Yaskawa INFORM job: TEST_KR.JBI

/JOB
//NAME TEST_KR
///FOLDERNAME INNE
//POS
///NPOS 2,2,0,0,0,0
///TOOL 0
///POSTYPE ROBOT
///RECTAN
///RCONF 0,0,0,0,0,0,0,0,0,0,0,0,0,0,0,0,0,0,0,0,0,0,0,0
C00000=-1082.109,-1268.604,-1687.249,-50.7166,43.0014,-29.7739
C00001=-1082.109,-1268.604,-1687.249,-50.7166,43.0014,-29.7739
BC00000=2160.163,372.281,1842.609
BC00001=2160.163,372.281,1842.609
//INST
///DATE 2023/10/04 15:12
///ATTR SC,RW,RJ
////FRAME ROBOT
///GROUP1 RB1,BS1
NOP
MOVJ C00000 BC00000 VJ=B000
MOVL C00001 BC00001 V=B001
END
